TYPE AX5000_S_0161 :
STRUCT
	Acceleration_data_scaling_factor:UINT;
END_STRUCT
END_TYPE

(* stored: Version 1.1.0.1, ProductVersion 3.1.4024.3
   DUT AX5000_S_0161: Id {55756622-86f7-44da-a837-19b7f463eff9} *)
